INTERFACE I_Car

METHOD PUBLIC ShowDetails : STRING
END_METHOD

END_INTERFACE

(* stored: Version 1.1.0.1, ProductVersion 3.1.4024.12
   Itf I_Car: Id {1b96b8e8-9a65-49bb-8085-4bf3ad7410e1}
   Method ShowDetails: Id {cf005e4d-18a0-4fd2-912e-9e852cc9ebf7} *)
